{attribute 'linkalways'} 
{attribute 'no_explicit_call' := 'This FB is a CLASS and must be accessed using methods or properties'}
{attribute 'enable_dynamic_creation'}
FUNCTION_BLOCK _ETcVnRotationAngle EXTENDS EnumDatatypeBase
VAR
	localData : ETcVnRotationAngle;
	activeData : REFERENCE TO ETcVnRotationAngle;
	enumBaseDatatype : _DINT(localData);
END_VAR

METHOD PRIVATE AddLocalEnumeration
VAR_INPUT
	Enumeration : T_MAXSTRING;
	Value : ETcVnRotationAngle;
END_VAR
AddEnumeration(Enumeration, Value);
END_METHOD

PROPERTY PUBLIC Address : PVOID
GET
Address := ADR(activeData);
END_GET
END_PROPERTY

METHOD PUBLIC ClearReference
VAR_INPUT
END_VAR
activeData REF= localData;
SetBaseDatatypeReference();
END_METHOD

METHOD PUBLIC Clone : I_Datatype
VAR
    pClone : POINTER TO _ETcVnRotationAngle;
END_VAR
pClone := __NEW(_ETcVnRotationAngle(InitialValue := Value));
Clone := pClone^;
END_METHOD

METHOD FB_init : BOOL
VAR_INPUT
	bInitRetains : BOOL; // if TRUE, the retain variables are initialized (warm start / cold start)
	bInCopyCode : BOOL;  // if TRUE, the instance afterwards gets moved into the copy code (online change)
	InitialValue : ETcVnRotationAngle;
END_VAR
localData := InitialValue;
AddBaseDatatype(enumBaseDatatype);
ClearReference();

AddLocalEnumeration('TCVN_RA_90_DEG', ETcVnRotationAngle.TCVN_RA_90_DEG);
AddLocalEnumeration('TCVN_RA_180_DEG', ETcVnRotationAngle.TCVN_RA_180_DEG);
AddLocalEnumeration('TCVN_RA_270_DEG', ETcVnRotationAngle.TCVN_RA_270_DEG);
END_METHOD

PROPERTY PUBLIC Identifier : T_MAXSTRING
GET
Identifier := 'ETcVnRotationAngle';
END_GET
END_PROPERTY

METHOD IsEnumeratorValueEqual : BOOL
VAR_INPUT
	Enumerator : I_KeyValueForwardEnumerator;
END_VAR
VAR
	storedValue : ETcVnRotationAngle;
END_VAR
IF NOT Enumerator.TryGet(storedValue) THEN
	RETURN;
END_IF

IsEnumeratorValueEqual := storedValue = activeData;
END_METHOD

METHOD PUBLIC MakeReferenceTo
VAR_INPUT
	ReferenceTarget : REFERENCE TO ETcVnRotationAngle;
END_VAR
activeData REF= ReferenceTarget;
SetBaseDatatypeReference();
END_METHOD

METHOD PROTECTED SetBaseDatatypeReference
VAR_INPUT
END_VAR
enumBaseDatatype.MakeReferenceTo(activeData);
END_METHOD

PROPERTY PUBLIC Size : UDINT
GET
Size := SIZEOF(activeData);
END_GET
END_PROPERTY

METHOD TryMakeReferenceTo : BOOL
VAR_INPUT
	Target : I_Datatype;
END_VAR
VAR
	targetAsEnum : I_EnumDatatype;
	pTargetData : POINTER TO ETcVnRotationAngle;
END_VAR
IF NOT Target.TryResolveAsEnumDatatype(targetAsEnum) THEN
	RETURN;
END_IF

IF targetAsEnum.Identifier <> Identifier THEN
	RETURN;
END_IF

pTargetData := Target.Address;
activeData REF= pTargetData^;
SetBaseDatatypeReference();
TryMakeReferenceTo := TRUE;
END_METHOD

PROPERTY PUBLIC Value : ETcVnRotationAngle
GET
Value := activeData;
END_GET
SET
activeData := Value;
END_SET
END_PROPERTY

END_FUNCTION_BLOCK

(* stored: Version 1.1.0.1, ProductVersion 3.1.4024.12
   POU _ETcVnRotationAngle: Id {a4de0f37-603e-452f-b5a3-eef93fd82d55}, SpecialFunc None
   Folder Constructor: Id {c3e45780-3b13-414b-bc95-e34c56b39977}
   Folder Private: Id {3911f586-c5ff-44b8-98c3-f8ee9ff356f4}
   Folder Protected: Id {7b1eef7f-6150-4ee4-9b6a-572bc468faad}
   Method AddLocalEnumeration: Id {78b081d6-f2b6-48fd-88da-1423baf65759}
   Property Address: Id {dad4f431-db95-4c34-90c2-062ffe180287}
   Get Get: Id {f01a71d1-06e0-4974-9906-a7b8f55bc39f}
   Method ClearReference: Id {0911fb67-8c76-4ee0-b344-92afef1d7725}
   Method Clone: Id {92d729a2-52e0-4e9b-af48-466d723316c0}
   Method FB_init: Id {ff01265b-eeef-48e4-ac10-028095bef40b}
   Property Identifier: Id {4d46b2eb-9bda-4c11-b26f-997e8d4b86dd}
   Get Get: Id {c8c4913c-d79f-431d-8e64-6fa9ebb1dc03}
   Method IsEnumeratorValueEqual: Id {77e96a17-f152-49f3-9ef5-8b56848d028b}
   Method MakeReferenceTo: Id {b578bdb9-bcef-4ab6-b259-7a6fc3325dfb}
   Method SetBaseDatatypeReference: Id {0716e2b2-c9be-446e-a9de-68c60d3c50ff}
   Property Size: Id {4c1e42b6-17b5-4dd7-aa97-db074466767c}
   Get Get: Id {e085c32e-e435-448e-8693-bb757cb4f703}
   Method TryMakeReferenceTo: Id {b37782c5-8bd0-4a09-97f6-3033d4276347}
   Property Value: Id {48318849-2cec-4ef1-a1cb-7bae000f1695}
   Get Get: Id {568302c2-7fd3-419c-8fb4-3788bf3bb033}
   Set Set: Id {014e4182-c7f0-49ed-a253-0d7110c8bcd3} *)
